(* CODESYS project 3.project

Project tree, tasks and I/O mapping:
  Device : CODESYS Control Win V3, 3S - Smart Software Solutions GmbH, order no. 305021, version 3.5.11.30
    application Application
      libraries: Standard, * (System)
      task MainTask (cyclic, interval t#20ms, priority 1) calls PLC_PRG
      program PLC_PRG [LD]
*)

// Device/Application/PLC_PRG
PROGRAM PLC_PRG
VAR
	BT1: BOOL;
	TOF_0: TOF;
	K3: BOOL;
	BT2: BOOL;
	K2: BOOL;
	K1: BOOL;
END_VAR

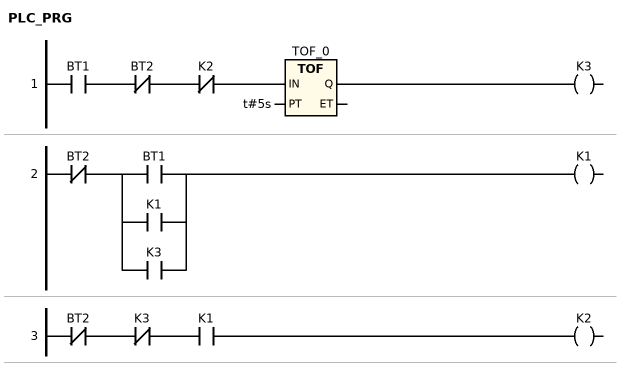
// NETWORK 1
TOF_0(IN := BT1 AND NOT BT2 AND NOT K2, PT := t#5s); // TOF
K3 := TOF_0.Q;

// NETWORK 2
K1 := NOT BT2 AND (BT1 OR K1 OR K3);

// NETWORK 3
K2 := NOT BT2 AND NOT K3 AND K1;

END_PROGRAM
